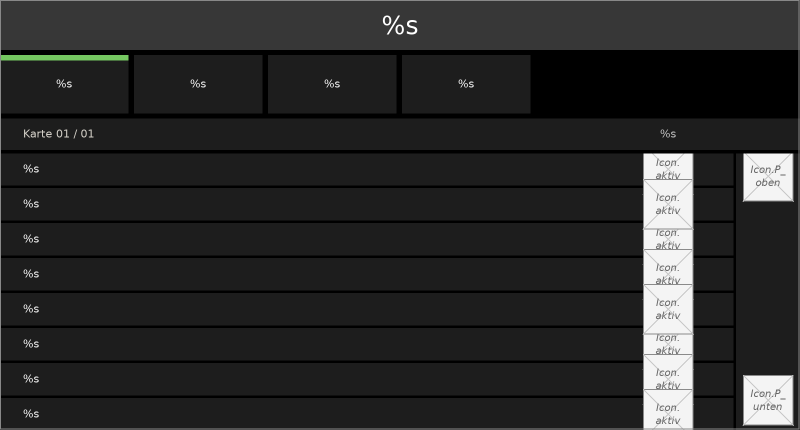
VISUALIZATION IO_Auswahl  // 800x430
    Frame (0,0 800x430), frame switch variable: Visu.i_Frame_Index
        shows Liste_DI()
        shows Liste_DO()
        shows Liste_AI()
        shows Liste_AO()
        shows SW_IBN_Einstellungen_K(i_titel := 69)
    Frame (0,430 800x50)
        shows Fusszeile_50()
END_VISUALIZATION

// ZY_Visu/IBN/Liste_AI
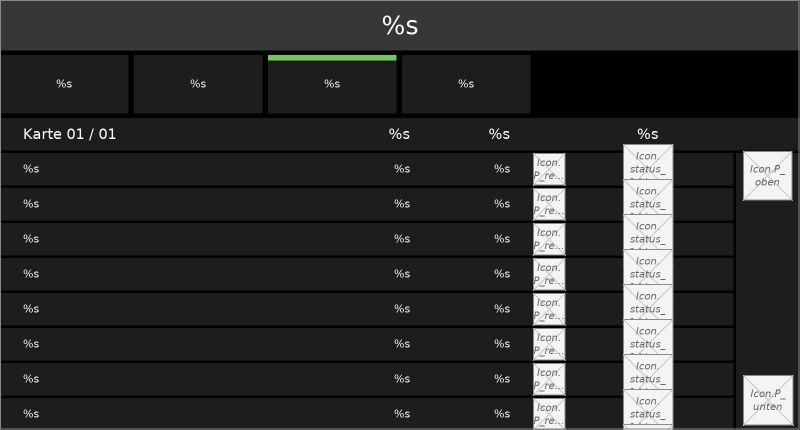
VISUALIZATION Liste_AI  // 800x430
    Rectangle (736,153 64x277)
    Image (743,375 50x50), image: Icon.P_unten
        OnMouseClick: execute {  }
    Image (743,151 49x49), image: Icon.P_oben
    Rectangle (0,153 733x32)
    Rectangle (20,153 400x32), "%s"
    Rectangle (0,223 733x32)
    Rectangle (20,223 400x32), "%s"
    Rectangle (0,188 733x32)
    Rectangle (20,188 400x32), "%s"
    Rectangle (0,258 733x32)
    Rectangle (20,258 400x32), "%s"
    Rectangle (0,328 733x32)
    Rectangle (20,328 400x32), "%s"
    Rectangle (0,293 733x32)
    Rectangle (20,293 400x32), "%s"
    Rectangle (0,538 733x32)
    Rectangle (20,538 400x32), "%s"
    Rectangle (0,363 733x32)
    Rectangle (20,363 400x32), "%s"
    Rectangle (0,433 733x32)
    Rectangle (20,433 400x32), "%s"
    Rectangle (0,398 733x32)
    Rectangle (20,398 400x32), "%s"
    Rectangle (0,468 733x32)
    Rectangle (20,468 400x32), "%s"
    Rectangle (0,503 733x32)
    Rectangle (20,503 400x32), "%s"
    Rectangle (0,118 800x32)
    Rectangle (20,118 324x32), "Karte 01 / 01"
    Rectangle (623,118 50x32), "%s", text list: 'Sprachen', text index: 49
    Image (623,144 50x50), image: Icon.status_fehlerfrei_element
    Image (623,144 50x50), image: Icon.status_fehler_element
    Image (533,153 32x32), image: Icon.P_rechts
        OnMouseClick: execute { Visu.i_Frame_Index:=4; }
    Rectangle (433,153 80x32), "%s"
    Rectangle (333,153 80x32), "%s"
    Rectangle (433,118 80x32), "%s", text list: 'Sprachen', text index: 50
    Rectangle (333,118 80x32), "%s", text list: 'Sprachen', text index: 51
    Image (623,179 50x50), image: Icon.status_fehlerfrei_element
    Image (623,179 50x50), image: Icon.status_fehler_element
    Image (533,188 32x32), image: Icon.P_rechts
    Rectangle (433,188 80x32), "%s"
    Rectangle (333,188 80x32), "%s"
    Image (623,214 50x50), image: Icon.status_fehlerfrei_element
    Image (623,214 50x50), image: Icon.status_fehler_element
    Image (533,223 32x32), image: Icon.P_rechts
    Rectangle (433,223 80x32), "%s"
    Rectangle (333,223 80x32), "%s"
    Image (623,249 50x50), image: Icon.status_fehlerfrei_element
    Image (623,249 50x50), image: Icon.status_fehler_element
    Image (533,258 32x32), image: Icon.P_rechts
    Rectangle (433,258 80x32), "%s"
    Rectangle (333,258 80x32), "%s"
    Image (623,284 50x50), image: Icon.status_fehlerfrei_element
    Image (623,284 50x50), image: Icon.status_fehler_element
    Image (533,293 32x32), image: Icon.P_rechts
    Rectangle (433,293 80x32), "%s"
    Rectangle (333,293 80x32), "%s"
    Image (623,319 50x50), image: Icon.status_fehlerfrei_element
    Image (623,319 50x50), image: Icon.status_fehler_element
    Image (533,328 32x32), image: Icon.P_rechts
    Rectangle (433,328 80x32), "%s"
    Rectangle (333,328 80x32), "%s"
    Image (623,354 50x50), image: Icon.status_fehlerfrei_element
    Image (623,354 50x50), image: Icon.status_fehler_element
    Image (533,363 32x32), image: Icon.P_rechts
    Rectangle (433,363 80x32), "%s"
    Rectangle (333,363 80x32), "%s"
    Image (623,389 50x50), image: Icon.status_fehlerfrei_element
    Image (623,389 50x50), image: Icon.status_fehler_element
    Image (533,398 32x32), image: Icon.P_rechts
    Rectangle (433,398 80x32), "%s"
    Rectangle (333,398 80x32), "%s"
    Image (623,424 50x50), image: Icon.status_fehlerfrei_element
    Image (623,424 50x50), image: Icon.status_fehler_element
    Image (533,433 32x32), image: Icon.P_rechts
    Rectangle (433,433 80x32), "%s"
    Rectangle (333,433 80x32), "%s"
    Image (623,459 50x50), image: Icon.status_fehlerfrei_element
    Image (623,459 50x50), image: Icon.status_fehler_element
    Image (533,468 32x32), image: Icon.P_rechts
    Rectangle (433,468 80x32), "%s"
    Rectangle (333,468 80x32), "%s"
    Image (623,494 50x50), image: Icon.status_fehlerfrei_element
    Image (623,494 50x50), image: Icon.status_fehler_element
    Image (533,503 32x32), image: Icon.P_rechts
    Rectangle (433,503 80x32), "%s"
    Rectangle (333,503 80x32), "%s"
    Image (623,529 50x50), image: Icon.status_fehlerfrei_element
    Image (623,529 50x50), image: Icon.status_fehler_element
    Image (533,538 32x32), image: Icon.P_rechts
    Rectangle (433,538 80x32), "%s"
    Rectangle (333,538 80x32), "%s"
    Rectangle (0,0 800x50), "%s", text list: 'Sprachen', text index: 44
    Rectangle (0,55 128x58), "%s", text list: 'Sprachen', text index: 45
        OnMouseClick: execute { Visu.i_Frame_Index:=0; }
    Rectangle (134,55 128x58), "%s", text list: 'Sprachen', text index: 46
        OnMouseClick: execute { Visu.i_Frame_Index:=1; }
    Rectangle (268,55 128x58), "%s", text list: 'Sprachen', text index: 47
        OnMouseClick: execute { Visu.i_Frame_Index:=2; }
    Rectangle (402,55 128x58), "%s", text list: 'Sprachen', text index: 48
        OnMouseClick: execute { Visu.i_Frame_Index:=3; }
    Rectangle (0,55 128x5)
    Rectangle (134,55 128x5)
    Rectangle (268,55 128x5)
    Rectangle (402,55 128x5)
END_VISUALIZATION

// ZY_Visu/IBN/Liste_AO
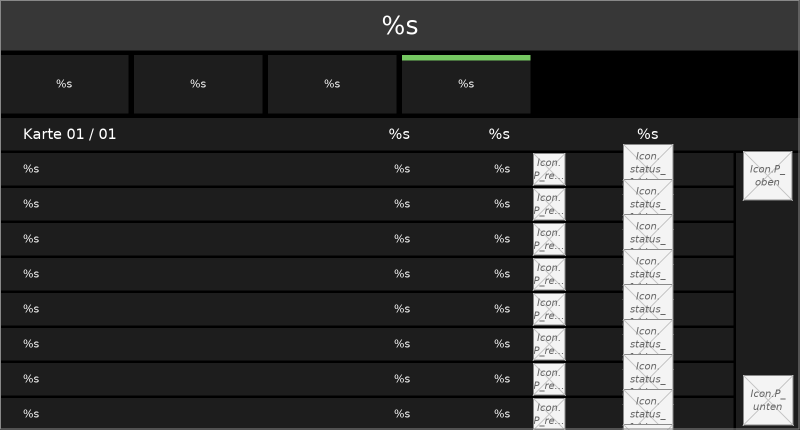
VISUALIZATION Liste_AO  // 800x430
    Rectangle (736,153 64x277)
    Image (743,375 50x50), image: Icon.P_unten
        OnMouseClick: execute {  }
    Image (743,151 49x49), image: Icon.P_oben
    Rectangle (0,153 733x32)
    Rectangle (20,153 400x32), "%s"
    Rectangle (0,223 733x32)
    Rectangle (20,223 400x32), "%s"
    Rectangle (0,188 733x32)
    Rectangle (20,188 400x32), "%s"
    Rectangle (0,258 733x32)
    Rectangle (20,258 400x32), "%s"
    Rectangle (0,328 733x32)
    Rectangle (20,328 400x32), "%s"
    Rectangle (0,293 733x32)
    Rectangle (20,293 400x32), "%s"
    Rectangle (0,538 733x32)
    Rectangle (20,538 400x32), "%s"
    Rectangle (0,363 733x32)
    Rectangle (20,363 400x32), "%s"
    Rectangle (0,433 733x32)
    Rectangle (20,433 400x32), "%s"
    Rectangle (0,398 733x32)
    Rectangle (20,398 400x32), "%s"
    Rectangle (0,468 733x32)
    Rectangle (20,468 400x32), "%s"
    Rectangle (0,503 733x32)
    Rectangle (20,503 400x32), "%s"
    Rectangle (0,118 800x32)
    Rectangle (20,118 324x32), "Karte 01 / 01"
    Rectangle (623,118 50x32), "%s", text list: 'Sprachen', text index: 49
    Image (623,144 50x50), image: Icon.status_fehlerfrei_element
    Image (623,144 50x50), image: Icon.status_fehler_element
    Image (533,153 32x32), image: Icon.P_rechts
        OnMouseClick: execute { Visu.i_Frame_Index:=4; }
    Rectangle (433,153 80x32), "%s"
    Rectangle (333,153 80x32), "%s"
    Rectangle (433,118 80x32), "%s", text list: 'Sprachen', text index: 50
    Rectangle (333,118 80x32), "%s", text list: 'Sprachen', text index: 51
    Image (623,179 50x50), image: Icon.status_fehlerfrei_element
    Image (623,179 50x50), image: Icon.status_fehler_element
    Image (533,188 32x32), image: Icon.P_rechts
    Rectangle (433,188 80x32), "%s"
    Rectangle (333,188 80x32), "%s"
    Image (623,214 50x50), image: Icon.status_fehlerfrei_element
    Image (623,214 50x50), image: Icon.status_fehler_element
    Image (533,223 32x32), image: Icon.P_rechts
    Rectangle (433,223 80x32), "%s"
    Rectangle (333,223 80x32), "%s"
    Image (623,249 50x50), image: Icon.status_fehlerfrei_element
    Image (623,249 50x50), image: Icon.status_fehler_element
    Image (533,258 32x32), image: Icon.P_rechts
    Rectangle (433,258 80x32), "%s"
    Rectangle (333,258 80x32), "%s"
    Image (623,284 50x50), image: Icon.status_fehlerfrei_element
    Image (623,284 50x50), image: Icon.status_fehler_element
    Image (533,293 32x32), image: Icon.P_rechts
    Rectangle (433,293 80x32), "%s"
    Rectangle (333,293 80x32), "%s"
    Image (623,319 50x50), image: Icon.status_fehlerfrei_element
    Image (623,319 50x50), image: Icon.status_fehler_element
    Image (533,328 32x32), image: Icon.P_rechts
    Rectangle (433,328 80x32), "%s"
    Rectangle (333,328 80x32), "%s"
    Image (623,354 50x50), image: Icon.status_fehlerfrei_element
    Image (623,354 50x50), image: Icon.status_fehler_element
    Image (533,363 32x32), image: Icon.P_rechts
    Rectangle (433,363 80x32), "%s"
    Rectangle (333,363 80x32), "%s"
    Image (623,389 50x50), image: Icon.status_fehlerfrei_element
    Image (623,389 50x50), image: Icon.status_fehler_element
    Image (533,398 32x32), image: Icon.P_rechts
    Rectangle (433,398 80x32), "%s"
    Rectangle (333,398 80x32), "%s"
    Image (623,424 50x50), image: Icon.status_fehlerfrei_element
    Image (623,424 50x50), image: Icon.status_fehler_element
    Image (533,433 32x32), image: Icon.P_rechts
    Rectangle (433,433 80x32), "%s"
    Rectangle (333,433 80x32), "%s"
    Image (623,459 50x50), image: Icon.status_fehlerfrei_element
    Image (623,459 50x50), image: Icon.status_fehler_element
    Image (533,468 32x32), image: Icon.P_rechts
    Rectangle (433,468 80x32), "%s"
    Rectangle (333,468 80x32), "%s"
    Image (623,494 50x50), image: Icon.status_fehlerfrei_element
    Image (623,494 50x50), image: Icon.status_fehler_element
    Image (533,503 32x32), image: Icon.P_rechts
    Rectangle (433,503 80x32), "%s"
    Rectangle (333,503 80x32), "%s"
    Image (623,529 50x50), image: Icon.status_fehlerfrei_element
    Image (623,529 50x50), image: Icon.status_fehler_element
    Image (533,538 32x32), image: Icon.P_rechts
    Rectangle (433,538 80x32), "%s"
    Rectangle (333,538 80x32), "%s"
    Rectangle (0,0 800x50), "%s", text list: 'Sprachen', text index: 44
    Rectangle (0,55 128x58), "%s", text list: 'Sprachen', text index: 45
        OnMouseClick: execute { Visu.i_Frame_Index:=0; }
    Rectangle (134,55 128x58), "%s", text list: 'Sprachen', text index: 46
        OnMouseClick: execute { Visu.i_Frame_Index:=1; }
    Rectangle (268,55 128x58), "%s", text list: 'Sprachen', text index: 47
        OnMouseClick: execute { Visu.i_Frame_Index:=2; }
    Rectangle (402,55 128x58), "%s", text list: 'Sprachen', text index: 48
        OnMouseClick: execute { Visu.i_Frame_Index:=3; }
    Rectangle (0,55 128x5)
    Rectangle (134,55 128x5)
    Rectangle (268,55 128x5)
    Rectangle (402,55 128x5)
END_VISUALIZATION

// ZY_Visu/IBN/Liste_DI
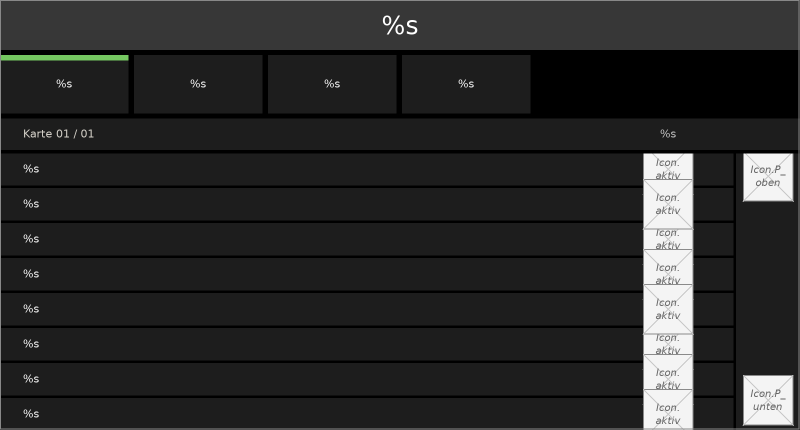
VISUALIZATION Liste_DI  // 800x430
VAR_IN_OUT

END_VAR
VAR
	i_verschieben:INT;


END_VAR
    Rectangle (736,153 64x277)
    Image (743,375 50x50), image: Icon.P_unten
        OnMouseClick: execute {
            IF i_verschieben<0 THEN
            	i_verschieben:=i_verschieben+35;
            End_if
        }
    Rectangle (0,153 733x32)
    Rectangle (0,223 733x32)
    Rectangle (0,188 733x32)
    Rectangle (0,258 733x32)
    Rectangle (0,328 733x32)
    Rectangle (0,293 733x32)
    Rectangle (0,538 733x32)
    Rectangle (0,363 733x32)
    Rectangle (0,433 733x32)
    Rectangle (0,398 733x32)
    Rectangle (0,468 733x32)
    Rectangle (0,503 733x32)
    Rectangle (20,153 400x32), "%s"
    Image (643,144 50x50), image: Icon.inaktiv
    Image (643,144 50x50), image: Icon.aktiv
    Rectangle (20,223 400x32), "%s"
    Image (643,214 50x50), image: Icon.inaktiv
    Image (643,214 50x50), image: Icon.aktiv
    Rectangle (20,188 400x32), "%s"
    Image (643,179 50x50), image: Icon.inaktiv
    Image (643,179 50x50), image: Icon.aktiv
    Rectangle (20,258 400x32), "%s"
    Image (643,249 50x50), image: Icon.inaktiv
    Image (643,249 50x50), image: Icon.aktiv
    Rectangle (20,328 400x32), "%s"
    Image (643,319 50x50), image: Icon.inaktiv
    Image (643,319 50x50), image: Icon.aktiv
    Rectangle (20,293 400x32), "%s"
    Image (643,284 50x50), image: Icon.inaktiv
    Image (643,284 50x50), image: Icon.aktiv
    Rectangle (20,538 400x32), "%s"
    Image (643,529 50x50), image: Icon.inaktiv
    Image (643,529 50x50), image: Icon.aktiv
    Rectangle (20,363 400x32), "%s"
    Image (643,354 50x50), image: Icon.inaktiv
    Image (643,354 50x50), image: Icon.aktiv
    Rectangle (20,433 400x32), "%s"
    Image (643,424 50x50), image: Icon.inaktiv
    Image (643,424 50x50), image: Icon.aktiv
    Rectangle (20,398 400x32), "%s"
    Image (643,389 50x50), image: Icon.inaktiv
    Image (643,389 50x50), image: Icon.aktiv
    Rectangle (20,468 400x32), "%s"
    Image (643,459 50x50), image: Icon.inaktiv
    Image (643,459 50x50), image: Icon.aktiv
    Rectangle (20,503 400x32), "%s"
    Image (643,494 50x50), image: Icon.inaktiv
    Image (643,494 50x50), image: Icon.aktiv
    Image (743,151 50x50), image: Icon.P_oben
        OnMouseClick: execute {
            IF  i_verschieben>-100 THEN
            	i_verschieben:=i_verschieben-35;
            End_if
        }
    Group (0,118 800x32)
        Rectangle (0,0 800x32)
        Rectangle (20,0 324x32), "Karte 01 / 01"
        Rectangle (643,0 50x32), "%s", text list: 'Sprachen', text index: 49
    Rectangle (0,0 800x50), "%s", text list: 'Sprachen', text index: 44
    Rectangle (0,50 800x68)
    Rectangle (0,55 128x58), "%s", text list: 'Sprachen', text index: 45
        OnMouseClick: execute { Visu.i_Frame_Index:=0; }
    Rectangle (134,55 128x58), "%s", text list: 'Sprachen', text index: 46
        OnMouseClick: execute { Visu.i_Frame_Index:=1; }
    Rectangle (268,55 128x58), "%s", text list: 'Sprachen', text index: 47
        OnMouseClick: execute { Visu.i_Frame_Index:=2; }
    Rectangle (402,55 128x58), "%s", text list: 'Sprachen', text index: 48
        OnMouseClick: execute { Visu.i_Frame_Index:=3; }
    Rectangle (0,55 128x5)
    Rectangle (0,150 800x3)
END_VISUALIZATION

// ZY_Visu/IBN/Liste_DO
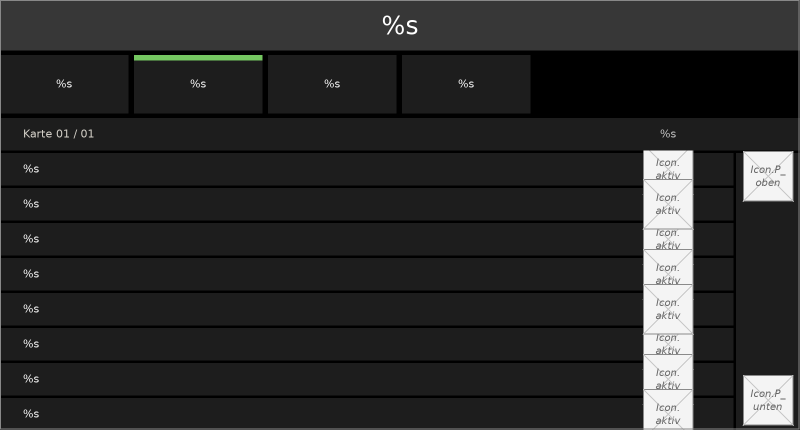
VISUALIZATION Liste_DO  // 800x430
    Rectangle (736,153 64x277)
    Image (743,375 50x50), image: Icon.P_unten
        OnMouseClick: execute {  }
    Image (743,151 50x50), image: Icon.P_oben
    Rectangle (0,153 733x32)
    Rectangle (0,223 733x32)
    Rectangle (0,188 733x32)
    Rectangle (0,258 733x32)
    Rectangle (0,328 733x32)
    Rectangle (0,293 733x32)
    Rectangle (0,538 733x32)
    Rectangle (0,363 733x32)
    Rectangle (0,433 733x32)
    Rectangle (0,398 733x32)
    Rectangle (0,468 733x32)
    Rectangle (0,503 733x32)
    Rectangle (20,153 400x32), "%s"
    Image (643,144 50x50), image: Icon.inaktiv
    Image (643,144 50x50), image: Icon.aktiv
    Rectangle (20,223 400x32), "%s"
    Image (643,214 50x50), image: Icon.inaktiv
    Image (643,214 50x50), image: Icon.aktiv
    Rectangle (20,188 400x32), "%s"
    Image (643,179 50x50), image: Icon.inaktiv
    Image (643,179 50x50), image: Icon.aktiv
    Rectangle (20,258 400x32), "%s"
    Image (643,249 50x50), image: Icon.inaktiv
    Image (643,249 50x50), image: Icon.aktiv
    Rectangle (20,328 400x32), "%s"
    Image (643,319 50x50), image: Icon.inaktiv
    Image (643,319 50x50), image: Icon.aktiv
    Rectangle (20,293 400x32), "%s"
    Image (643,284 50x50), image: Icon.inaktiv
    Image (643,284 50x50), image: Icon.aktiv
    Rectangle (20,538 400x32), "%s"
    Image (643,529 50x50), image: Icon.inaktiv
    Image (643,529 50x50), image: Icon.aktiv
    Rectangle (20,363 400x32), "%s"
    Image (643,354 50x50), image: Icon.inaktiv
    Image (643,354 50x50), image: Icon.aktiv
    Rectangle (20,433 400x32), "%s"
    Image (643,424 50x50), image: Icon.inaktiv
    Image (643,424 50x50), image: Icon.aktiv
    Rectangle (20,398 400x32), "%s"
    Image (643,389 50x50), image: Icon.inaktiv
    Image (643,389 50x50), image: Icon.aktiv
    Rectangle (20,468 400x32), "%s"
    Image (643,459 50x50), image: Icon.inaktiv
    Image (643,459 50x50), image: Icon.aktiv
    Rectangle (20,503 400x32), "%s"
    Image (643,494 50x50), image: Icon.inaktiv
    Image (643,494 50x50), image: Icon.aktiv
    Group (0,118 800x32)
        Rectangle (0,0 800x32)
        Rectangle (20,0 324x32), "Karte 01 / 01"
        Rectangle (643,0 50x32), "%s", text list: 'Sprachen', text index: 49
    Rectangle (0,0 800x50), "%s", text list: 'Sprachen', text index: 44
    Rectangle (0,55 128x58), "%s", text list: 'Sprachen', text index: 45
        OnMouseClick: execute { Visu.i_Frame_Index:=0; }
    Rectangle (134,55 128x58), "%s", text list: 'Sprachen', text index: 46
        OnMouseClick: execute { Visu.i_Frame_Index:=1; }
    Rectangle (268,55 128x58), "%s", text list: 'Sprachen', text index: 47
        OnMouseClick: execute { Visu.i_Frame_Index:=2; }
    Rectangle (402,55 128x58), "%s", text list: 'Sprachen', text index: 48
        OnMouseClick: execute { Visu.i_Frame_Index:=3; }
    Rectangle (0,55 128x5)
    Rectangle (134,55 128x5)
    Rectangle (268,55 128x5)
    Rectangle (402,55 128x5)
END_VISUALIZATION

// ZY_Visu/IBN/SW_IBN_Einstellungen_K
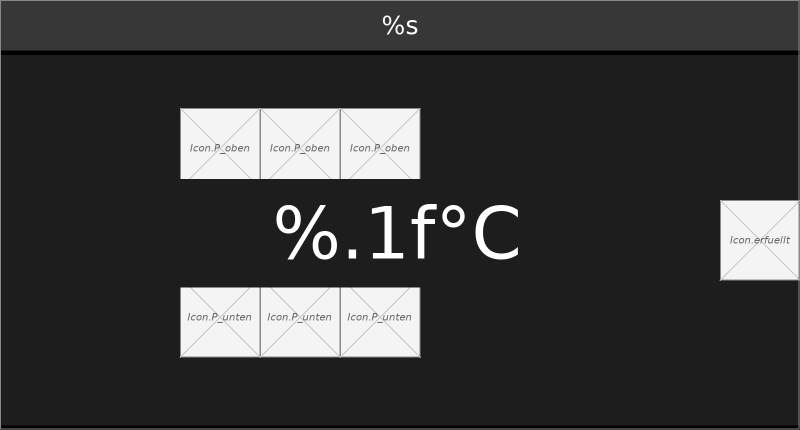
VISUALIZATION SW_IBN_Einstellungen_K  // 800x430
VAR_IN_OUT

END_VAR

VAR_INPUT
	i_titel:INT;
END_VAR
    Rectangle (0,0 800x50), "%s", text list: 'Sprachen', text index: i_titel
    Rectangle (0,55 800x370)
    Image (720,200 80x80), image: Icon.erfuellt
        OnMouseClick: execute { Visu.i_Frame_Index:=0; }
    Image (180,108 80x80), image: Icon.P_oben
    Image (180,277 80x80), image: Icon.P_unten
    Image (260,108 80x80), image: Icon.P_oben
    Image (340,108 80x80), image: Icon.P_oben
        OnMouseClick: execute {  }
    Image (260,277 80x80), image: Icon.P_unten
    Image (340,277 80x80), image: Icon.P_unten
    Rectangle (110,179 415x108), "%.1f°C"
END_VISUALIZATION

// ZY_Visu/Infoseite/Infoliste
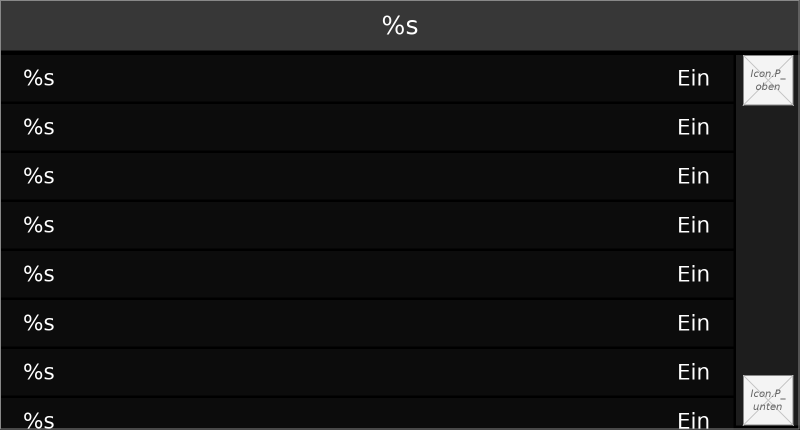
VISUALIZATION Infoliste  // 800x430
VAR_IN_OUT
	
END_VAR
VAR_INPUT
	i_Titel:INT;
	
END_VAR
VAR
	x_auf:BOOL;
	x_ab:BOOL;
	i_verschieben:INT:=0;
END_VAR
    Rectangle (0,0 800x50), "%s", text list: 'Sprachen', text index: i_Titel
    Rectangle (0,55 733x46)
    Label (20,55 479x46), "%s"
    Rectangle (0,104 733x46)
    Label (20,104 479x46), "%s"
    Rectangle (0,153 733x46)
    Label (20,153 479x46), "%s"
    Rectangle (0,202 733x46)
    Label (20,202 479x46), "%s"
    Rectangle (0,251 733x46)
    Label (20,251 479x46), "%s"
    Rectangle (0,300 733x46)
    Label (20,300 479x46), "%s"
    Rectangle (0,349 733x46)
    Label (20,349 479x46), "%s"
    Rectangle (583,55 130x46), "Ein"
    Rectangle (583,104 130x46), "Ein"
    Rectangle (0,398 733x46)
    Label (20,398 479x46), "%s"
    Rectangle (0,447 733x46)
    Label (20,447 479x46), "%s"
    Rectangle (0,496 733x46)
    Label (20,496 479x46), "%s"
    Rectangle (0,545 733x46)
    Label (20,545 479x46), "%s"
    Rectangle (583,545 130x46), "Ein"
    Rectangle (0,594 733x46)
    Label (20,594 479x46), "%s"
    Rectangle (583,153 130x46), "Ein"
    Rectangle (583,202 130x46), "Ein"
    Rectangle (583,251 130x46), "Ein"
    Rectangle (583,349 130x46), "Ein"
    Rectangle (583,300 130x46), "Ein"
    Rectangle (583,398 130x46), "Ein"
    Rectangle (583,447 130x46), "Ein"
    Rectangle (583,496 130x46), "Ein"
    Rectangle (583,594 130x46), "Ein"
    Group (736,55 64x370)
        Rectangle (0,0 64x370)
        Image (7,320 50x50), image: Icon.P_unten
            OnMouseClick:  ToggleVariable=x_ab
            OnMouseClick: execute {
                IF x_ab THEN
                	i_verschieben:=i_verschieben+50;
                	x_ab:=0;
                END_IF
            }
        Image (7,0 50x50), image: Icon.P_oben
            OnMouseClick:  ToggleVariable=x_auf
            OnMouseClick: execute {
                IF x_auf THEN
                	i_verschieben:=i_verschieben-50;
                	x_auf:=0;
                END_IF
            }
END_VISUALIZATION

// ZY_Visu/Infoseite/Infoseite
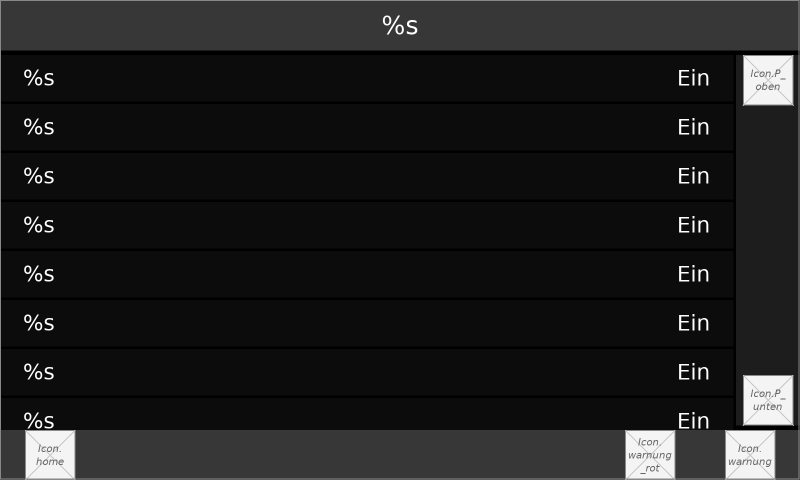
VISUALIZATION Infoseite  // 800x480
    Frame (0,0 800x430)
        shows Infoliste(i_Titel := 31)
    Frame (0,430 800x50)
        shows Fusszeile_50()
END_VISUALIZATION

// ZY_Visu/Sollwertmenu_9/Sollwerte Einstellungen/SW_Einstellungen_C
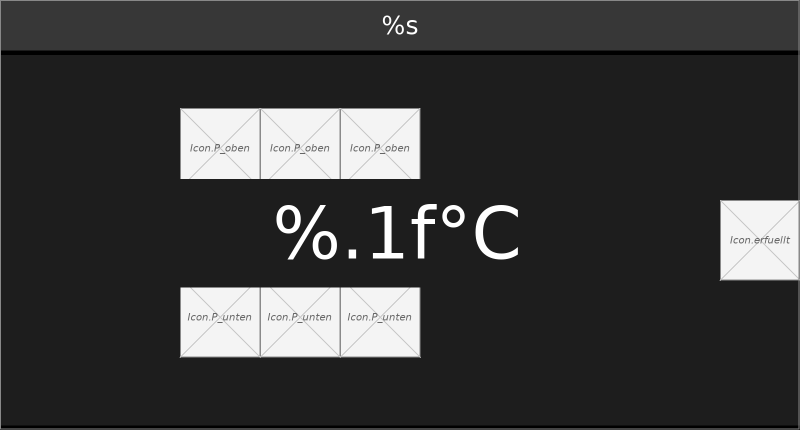
VISUALIZATION SW_Einstellungen_C  // 800x430
VAR_IN_OUT
		f_Data:REAL;
END_VAR

VAR_INPUT
	i_titel:INT;
END_VAR
    Rectangle (0,0 800x50), "%s", text list: 'Sprachen', text index: i_titel
    Rectangle (0,55 800x370), text variable: f_Data
    Image (720,200 80x80), image: Icon.erfuellt
        OnMouseClick: execute { Visu.i_Frame_Index:=0; }
    Image (180,108 80x80), image: Icon.P_oben
        OnMouseClick: execute { f_Data:=f_Data +10; }
    Image (180,277 80x80), image: Icon.P_unten
        OnMouseClick: execute { f_Data:=f_Data -10; }
    Image (260,108 80x80), image: Icon.P_oben
        OnMouseClick: execute { f_Data:=f_Data +1; }
    Image (340,108 80x80), image: Icon.P_oben
        OnMouseClick: execute { f_Data:=f_Data +0.1; }
    Image (260,277 80x80), image: Icon.P_unten
        OnMouseClick: execute { f_Data:=f_Data -1; }
    Image (340,277 80x80), image: Icon.P_unten
        OnMouseClick: execute { f_Data:=f_Data -0.1; }
    Rectangle (110,179 415x108), "%.1f°C", text variable: f_Data
END_VISUALIZATION

// ZY_Visu/Sollwertmenu_9/Sollwerte Einstellungen/SW_Einstellungen_Faktor
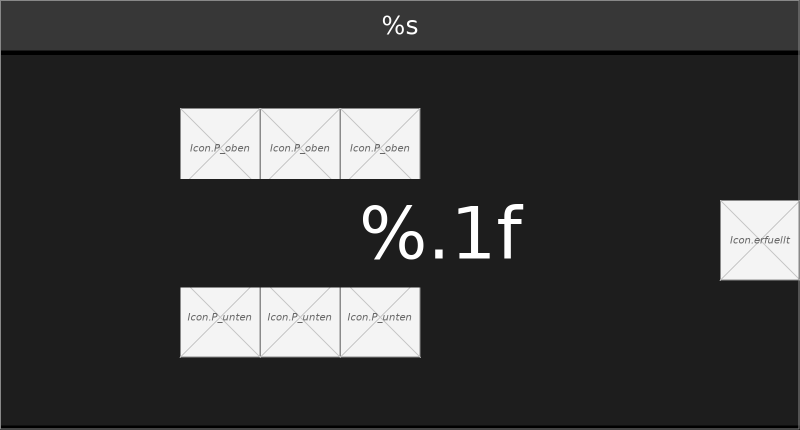
VISUALIZATION SW_Einstellungen_Faktor  // 800x430
VAR_IN_OUT
		f_Data:REAL;
END_VAR

VAR_INPUT
	i_titel:INT;
END_VAR
    Rectangle (0,0 800x50), "%s", text list: 'Sprachen', text index: i_titel
    Rectangle (0,55 800x370), text variable: f_Data
    Image (720,200 80x80), image: Icon.erfuellt
        OnMouseClick: execute { Visu.i_Frame_Index:=0; }
    Image (180,108 80x80), image: Icon.P_oben
        OnMouseClick: execute { f_Data:=f_Data +10; }
    Image (180,277 80x80), image: Icon.P_unten
        OnMouseClick: execute { f_Data:=f_Data -10; }
    Image (260,108 80x80), image: Icon.P_oben
        OnMouseClick: execute { f_Data:=f_Data +1; }
    Image (340,108 80x80), image: Icon.P_oben
        OnMouseClick: execute { f_Data:=f_Data +0.1; }
    Image (260,277 80x80), image: Icon.P_unten
        OnMouseClick: execute { f_Data:=f_Data -1; }
    Image (340,277 80x80), image: Icon.P_unten
        OnMouseClick: execute { f_Data:=f_Data -0.1; }
    Rectangle (110,179 415x108), "%.1f", text variable: f_Data
END_VISUALIZATION

// ZY_Visu/Sollwertmenu_9/Sollwerte Einstellungen/SW_Einstellungen_K
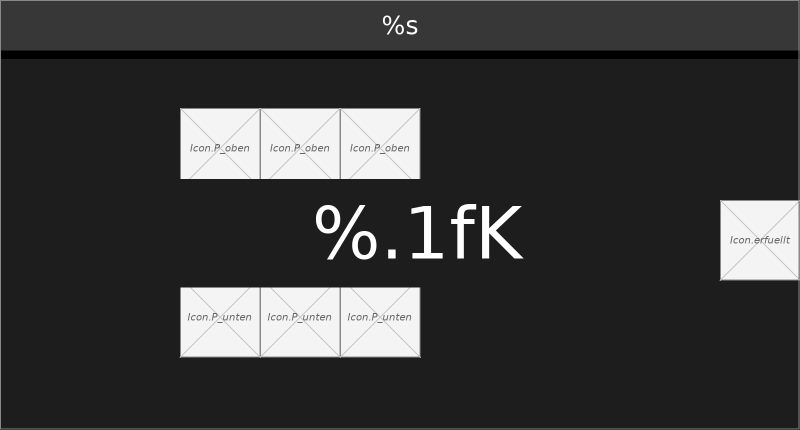
VISUALIZATION SW_Einstellungen_K  // 800x430
VAR_IN_OUT
		f_Data:REAL;
END_VAR

VAR_INPUT
	i_titel:INT;
END_VAR
    Rectangle (0,0 800x50), "%s", text list: 'Sprachen', text index: i_titel
    Rectangle (1,59 800x370), text variable: f_Data
    Image (720,200 80x80), image: Icon.erfuellt
        OnMouseClick: execute { Visu.i_Frame_Index:=0; }
    Image (180,108 80x80), image: Icon.P_oben
        OnMouseClick: execute { f_Data:=f_Data +10; }
    Image (180,277 80x80), image: Icon.P_unten
        OnMouseClick: execute { f_Data:=f_Data -10; }
    Image (260,108 80x80), image: Icon.P_oben
        OnMouseClick: execute { f_Data:=f_Data +1; }
    Image (340,108 80x80), image: Icon.P_oben
        OnMouseClick: execute { f_Data:=f_Data +0.1; }
    Image (260,277 80x80), image: Icon.P_unten
        OnMouseClick: execute { f_Data:=f_Data -1; }
    Image (340,277 80x80), image: Icon.P_unten
        OnMouseClick: execute { f_Data:=f_Data -0.1; }
    Rectangle (110,179 415x108), "%.1fK", text variable: f_Data
END_VISUALIZATION

// ZY_Visu/Sollwertmenu_9/Sollwerte Einstellungen/SW_Einstellungen_min
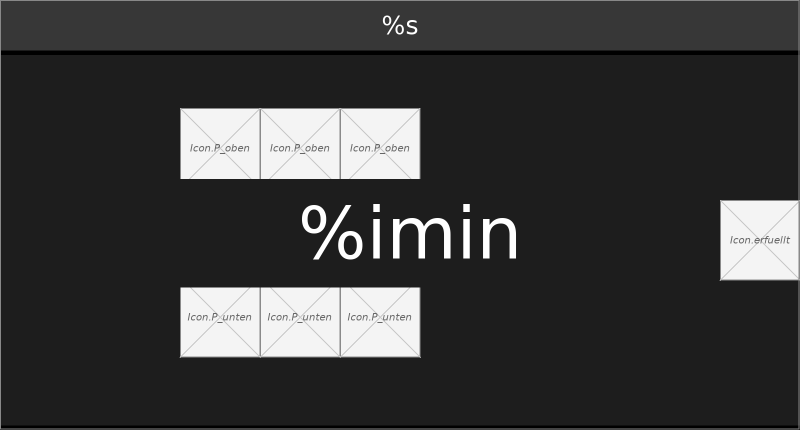
VISUALIZATION SW_Einstellungen_min  // 800x430
VAR_IN_OUT
		f_Data:WORD;
END_VAR

VAR_INPUT
	i_titel:INT;
END_VAR
    Rectangle (0,0 800x50), "%s", text list: 'Sprachen', text index: i_titel
    Rectangle (0,55 800x370), text variable: f_Data
    Image (720,200 80x80), image: Icon.erfuellt
        OnMouseClick: execute { Visu.i_Frame_Index:=0; }
    Image (180,108 80x80), image: Icon.P_oben
        OnMouseClick: execute { f_Data:=f_Data +10; }
    Image (180,277 80x80), image: Icon.P_unten
        OnMouseClick: execute { f_Data:=f_Data -10; }
    Image (260,108 80x80), image: Icon.P_oben
        OnMouseClick: execute { f_Data:=f_Data +1; }
    Image (340,108 80x80), image: Icon.P_oben
        OnMouseClick: execute { f_Data:=f_Data +0.1; }
    Image (260,277 80x80), image: Icon.P_unten
        OnMouseClick: execute { f_Data:=f_Data -1; }
    Image (340,277 80x80), image: Icon.P_unten
        OnMouseClick: execute { f_Data:=f_Data -0.1; }
    Rectangle (110,179 415x108), "%imin", text variable: f_Data
END_VISUALIZATION

// ZY_Visu/Sollwertmenu_9/Sollwerte Einstellungen/SW_Einstellungen_ms
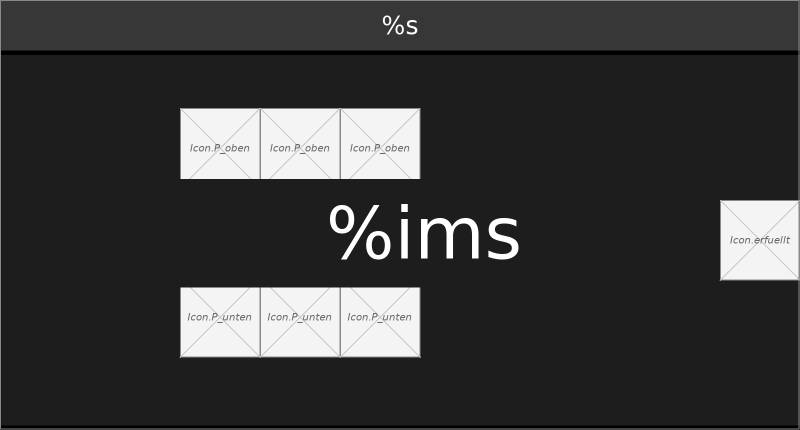
VISUALIZATION SW_Einstellungen_ms  // 800x430
VAR_IN_OUT
		f_Data:WORD;
END_VAR

VAR_INPUT
	i_titel:INT;
END_VAR
    Rectangle (0,0 800x50), "%s", text list: 'Sprachen', text index: i_titel
    Rectangle (0,55 800x370), text variable: f_Data
    Image (720,200 80x80), image: Icon.erfuellt
        OnMouseClick: execute { Visu.i_Frame_Index:=0; }
    Image (180,108 80x80), image: Icon.P_oben
        OnMouseClick: execute { f_Data:=f_Data +10; }
    Image (180,277 80x80), image: Icon.P_unten
        OnMouseClick: execute { f_Data:=f_Data -10; }
    Image (260,108 80x80), image: Icon.P_oben
        OnMouseClick: execute { f_Data:=f_Data +1; }
    Image (340,108 80x80), image: Icon.P_oben
        OnMouseClick: execute { f_Data:=f_Data +0.1; }
    Image (260,277 80x80), image: Icon.P_unten
        OnMouseClick: execute { f_Data:=f_Data -1; }
    Image (340,277 80x80), image: Icon.P_unten
        OnMouseClick: execute { f_Data:=f_Data -0.1; }
    Rectangle (110,179 415x108), "%ims", text variable: f_Data
END_VISUALIZATION

// ZY_Visu/Sollwertmenu_9/Sollwerte Einstellungen/SW_zuruecksetzen
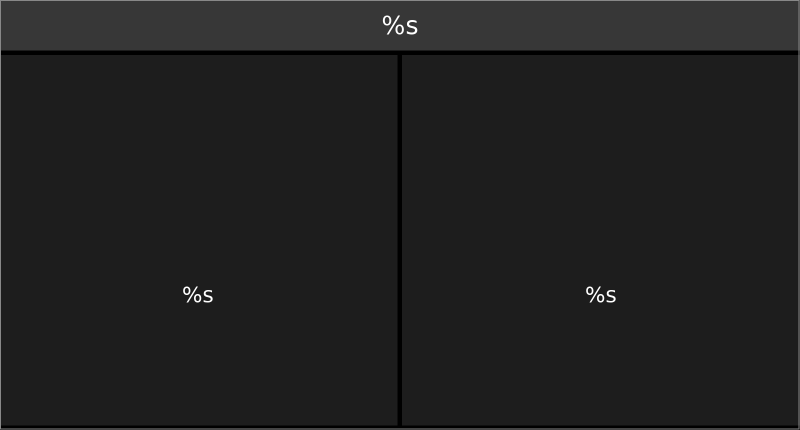
VISUALIZATION SW_zuruecksetzen  // 800x430
VAR_IN_OUT
	x_Zuruecksetzen:BOOL;
END_VAR

VAR_OUTPUT
	

END_VAR

VAR_INPUT
	i_Titel:INT;
	i_Text_1:INT;
	i_Text_2:INT;	

	
END_VAR
    Rectangle (0,0 800x50), "%s", text list: 'Sprachen', text index: i_Titel
    Rectangle (0,55 397x370)
        OnMouseClick: execute { Visu.i_Frame_Index:=0; }
    Rectangle (0,55 397x5)
    Rectangle (123,280 150x30), "%s", text list: 'Sprachen', text index: i_Text_1
    Polygon (943,131)
    Rectangle (402,55 398x370)
        OnMouseDown: execute { x_Zuruecksetzen:=TRUE; }
        OnMouseUp: execute { x_Zuruecksetzen:=false; }
    Rectangle (402,55 398x5)
    Rectangle (402,280 398x30), "%s", text list: 'Sprachen', text index: i_Text_2
END_VISUALIZATION

// ZY_Visu/Sollwertmenu_9/Sollwertmenu/Sollwertmenu
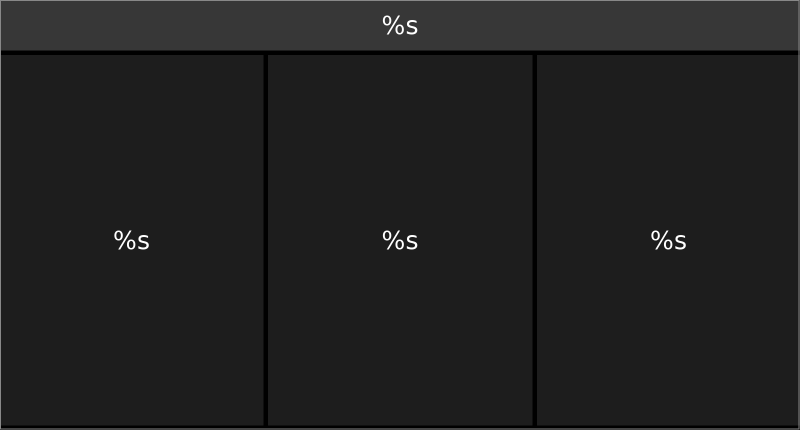
VISUALIZATION Sollwertmenu  // 800x430
    Rectangle (0,0 800x50), "%s", text list: 'Sprachen', text index: 3
    Rectangle (0,55 263x370), "%s", text list: 'Sprachen', text index: 0
        OnMouseClick:  Assign=Sollwertmenu_Waermegewinnung, Type=Assignment
    Rectangle (268,55 264x370), "%s", text list: 'Sprachen', text index: 1
        OnMouseClick:  Assign=Sollwertmenu_Waermepumpe, Type=Assignment
    Rectangle (537,55 263x370), "%s", text list: 'Sprachen', text index: 2
        OnMouseClick:  Assign=Sollwertmenu_Waermesenke, Type=Assignment
    Frame (0,430 800x50)
        shows Fusszeile_50()
    Image (125,430 50x50), image: Icon.zurueck
        OnMouseClick:  Assign=Hauptmenu, Type=Assignment
END_VISUALIZATION

// ZY_Visu/Sollwertmenu_9/Wärmegewinnung/UWP/SW_WG_UWP_Verd
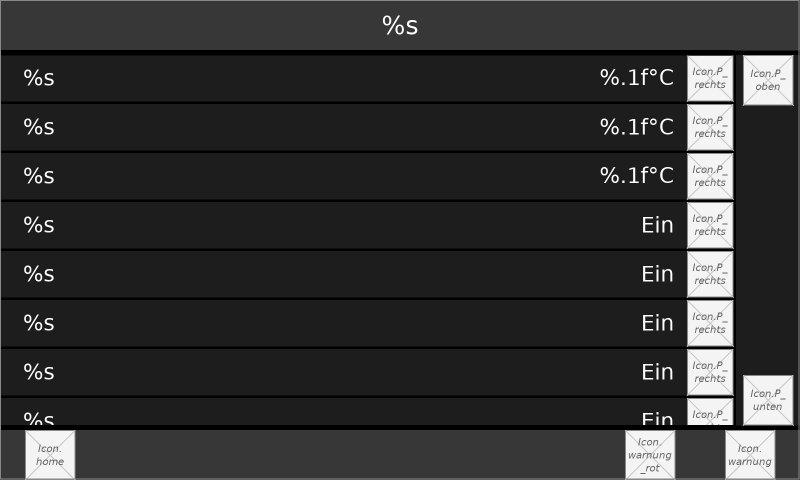
VISUALIZATION SW_WG_UWP_Verd  // 800x480
VAR_IN_OUT
	FB_GR2:GR_2;
END_VAR
    Frame (0,0 800x430), frame switch variable: GWP_Library.Visu.i_Frame_Index
        shows SW_WG_UWP_Verd_Liste(i_Titel := 25, FB_GR2 := FB_GR2)
        shows SW_Einstellungen_Zeit(i_titel := 53, f_Data := FB_GR2.f_AT)
        shows SW_Einstellungen_C(i_titel := 30, f_Data := FB_GR2.f_RefPunkt_TO1)
        shows SW_Einstellungen_C_1(i_titel := 31, f_Data := FB_GR2.f_SW_Min)
        shows SW_Einstellungen_Zeit(i_titel := 30)
    Frame (0,430 800x50)
        shows Fusszeile_50()
END_VISUALIZATION

// ZY_Visu/Sollwertmenu_9/Wärmegewinnung/UWP/SW_WG_UWP_Verd_Liste
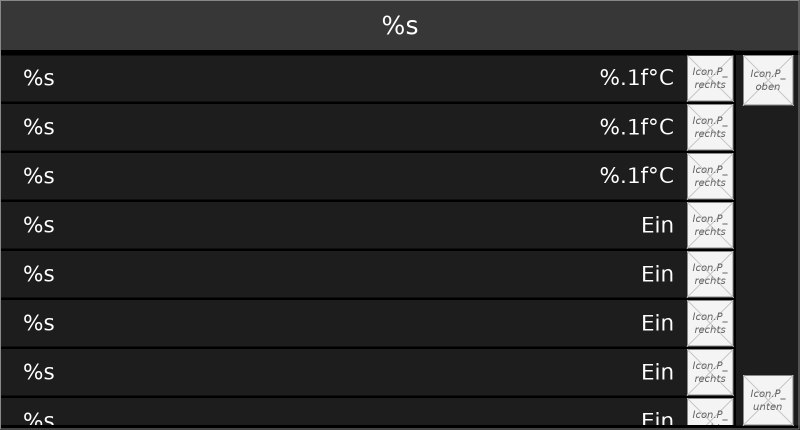
VISUALIZATION SW_WG_UWP_Verd_Liste  // 800x430
VAR_IN_OUT
	FB_GR2:GR_2;
END_VAR

VAR_INPUT
	i_Titel:INT;
END_VAR

VAR
	i_verschieben:INT;
 END_VAR
    Rectangle (0,55 733x46)
    Label (20,55 479x46), "%s"
    Rectangle (0,104 733x46)
    Label (20,104 479x46), "%s"
    Rectangle (547,55 130x45), "%.1f°C", text variable: FB_GR2.f_AT
    Rectangle (547,104 130x46), "%.1f°C", text variable: FB_GR2.f_RefPunkt_TO1
    Image (687,55 46x46), image: Icon.P_rechts
        OnMouseClick: execute { Visu.i_Frame_Index:=1; }
    Image (687,104 46x46), image: Icon.P_rechts
        OnMouseClick: execute { Visu.i_Frame_Index:=2; }
    Rectangle (0,153 733x46)
    Label (20,153 479x46), "%s"
    Rectangle (0,202 733x46)
    Label (20,202 479x46), "%s"
    Rectangle (0,251 733x46)
    Label (20,251 479x46), "%s"
    Rectangle (0,300 733x46)
    Label (20,300 479x46), "%s"
    Rectangle (0,349 733x46)
    Label (20,349 479x46), "%s"
    Rectangle (0,398 733x46)
    Label (20,398 479x46), "%s"
    Rectangle (0,447 733x46)
    Label (20,447 479x46), "%s"
    Rectangle (0,496 733x46)
    Label (20,496 479x46), "%s"
    Rectangle (0,545 733x46)
    Label (20,545 479x46), "%s"
    Rectangle (547,153 130x45), "%.1f°C", text variable: FB_GR2.f_SW_Min
        OnMouseClick: execute { GWP_Library.Visu.i_Frame_Index:=2; }
    Rectangle (547,202 130x46), "Ein"
    Rectangle (547,251 130x46), "Ein"
    Rectangle (547,300 130x46), "Ein"
    Rectangle (547,349 130x46), "Ein"
    Rectangle (547,447 130x46), "Ein"
    Rectangle (547,398 130x46), "Ein"
    Rectangle (547,496 130x46), "Ein"
    Rectangle (547,545 130x46), "Ein"
    Image (687,153 46x46), image: Icon.P_rechts
        OnMouseClick: execute { GWP_Library.Visu.i_Frame_Index:=3; }
    Image (687,545 46x46), image: s
    Image (687,496 46x46), image: Icon.P_rechts
    Image (687,447 46x46), image: Icon.P_rechts
    Image (687,398 46x46), image: Icon.P_rechts
    Image (687,349 46x46), image: Icon.P_rechts
    Image (687,300 46x46), image: Icon.P_rechts
    Image (687,251 46x46), image: Icon.P_rechts
    Image (687,202 46x46), image: Icon.P_rechts
    Rectangle (0,594 733x46)
    Label (20,594 479x46), "%s"
    Rectangle (547,594 130x45), "Ein"
    Image (687,594 46x46), image: Icon.P_rechts
    Image (79,430 50x50), image: Icon.zurueck
        OnMouseClick:  Assign=Sollwertmenu_Waermegewinnung, Type=Assignment
        OnMouseClick: execute { i_verschieben:=0; }
    Rectangle (0,0 800x50), "%s", text list: 'Sprachen', text index: i_Titel
    Group (736,55 64x370)
        Rectangle (0,0 64x370)
        Image (7,320 50x50), image: Icon.P_unten
            OnMouseClick: execute {
                IF i_verschieben<0 THEN
                	i_verschieben:=i_verschieben+53;
                End_if
            }
        Image (7,0 50x50), image: Icon.P_oben
            OnMouseClick: execute {
                IF  i_verschieben>-200 THEN
                	i_verschieben:=i_verschieben-53;
                End_if
            }
    Rectangle (0,50 733x5)
    Rectangle (0,425 733x5)
END_VISUALIZATION

// ZY_Visu/Sollwertmenu_9/Wärmegewinnung/Kachel_Abtauspeicher
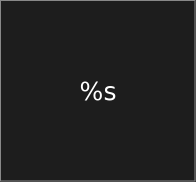
VISUALIZATION Kachel_Abtauspeicher  // 196x182
    Rectangle (0,0 196x182), "%s", text list: 'Sprachen', text index: 10
END_VISUALIZATION

// ZY_Visu/Sollwertmenu_9/Wärmegewinnung/Kachel_Abtauungen
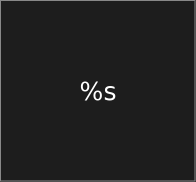
VISUALIZATION Kachel_Abtauungen  // 196x182
    Rectangle (0,0 196x182), "%s", text list: 'Sprachen', text index: 11
END_VISUALIZATION

// ZY_Visu/Sollwertmenu_9/Wärmegewinnung/Kachel_Abwaerme
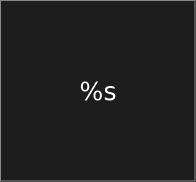
VISUALIZATION Kachel_Abwaerme  // 196x182
    Rectangle (0,0 196x182), "%s", text list: 'Sprachen', text index: 12
END_VISUALIZATION

// ZY_Visu/Sollwertmenu_9/Wärmegewinnung/Kachel_Erdsonden
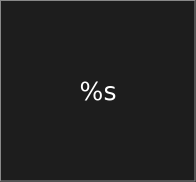
VISUALIZATION Kachel_Erdsonden  // 196x182
    Rectangle (0,0 196x182), "%s", text list: 'Sprachen', text index: 6
END_VISUALIZATION

// ZY_Visu/Sollwertmenu_9/Wärmegewinnung/Kachel_Grundwasser
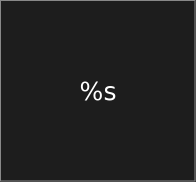
VISUALIZATION Kachel_Grundwasser  // 196x182
    Rectangle (0,0 196x182), "%s", text list: 'Sprachen', text index: 7
END_VISUALIZATION

// ZY_Visu/Sollwertmenu_9/Wärmegewinnung/Kachel_Luft
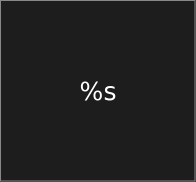
VISUALIZATION Kachel_Luft  // 196x182
    Rectangle (0,0 196x182), "%s", text list: 'Sprachen', text index: 8
END_VISUALIZATION

// ZY_Visu/Sollwertmenu_9/Wärmegewinnung/Kachel_Tiefhaltung
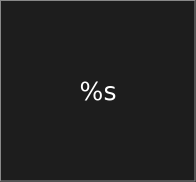
VISUALIZATION Kachel_Tiefhaltung  // 196x182
    Rectangle (0,0 196x182), "%s", text list: 'Sprachen', text index: 9
END_VISUALIZATION

// ZY_Visu/Sollwertmenu_9/Wärmegewinnung/Kachel_UWP_Verd
